Universal Robots PolyScope program: p1kine.urp

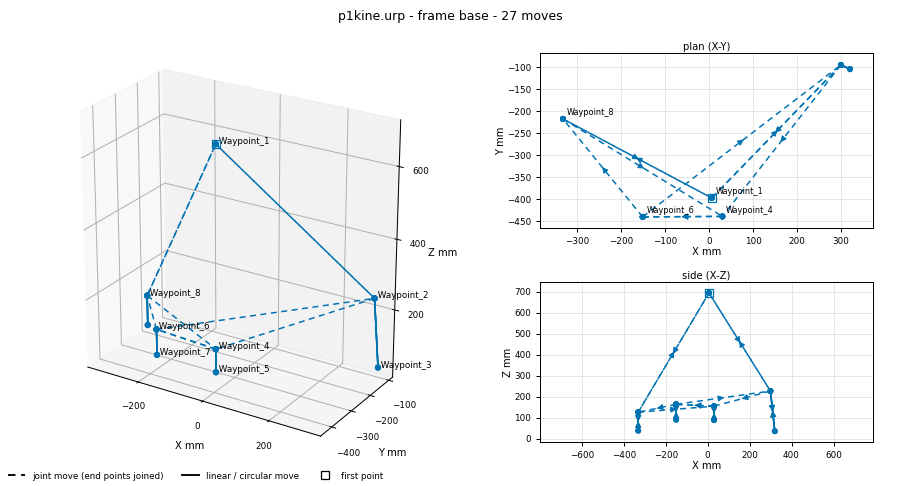
[picture p0: tool path of p1kine.urp in frame base, 27 of 27 moves have a stored position in this frame; points joined in program order, loops and branches not executed]
Program p1kine (installation=default directory=/programs createdIn=5.14.5 lastSavedIn=5.14.5 robotSerialNumber=20195300809)
Calibrated DH parameters: a=[-0.000085, -0.20076, -0.212369, 0.000121, -0.000118, 0]; d=[0.15185, -26.306375, 24.753047, 1.684739, 0.085386, 0.092088]; alpha=[1.572149, -0.00522, -0.011864, 1.571339, -1.571085, 0]; deltaTheta=[0, 0.599885, -0.513355, -0.086555, 0.000006, 0]
InitVariablesNode
Robot Program (runOnlyOnce=false)
  'Make sure gripper open'
  URCap Gripper Activate (Robotiq_Grippers, Robotiq Inc.) dataModel(ResetAndActivateKey=false)
  URCap Gripper (Robotiq_Grippers, Robotiq Inc.) dataModel(position=0.0, force=0.0, speed=100.0, positionInDouble=0.0, forceInDouble=0.0, speedInDouble=100.0, slaveIds=[9], blocking=true)
  Wait Sleep waitTime=1
  MoveJ speed 60 deg/s, acceleration 80 deg/s^2 (useActiveTCP=true) feature=Base
    Waypoint Waypoint_1: TCP in base x=6.371 y=-396.697 z=694.74 mm, rx=-0.018 ry=2.2102 rz=-2.2165 rad; joints [0.003, -90.002, 0, -90.003, 0.001, 0.002] deg; TCP offset x=0 y=0 z=174 mm, rx=0 ry=0 rz=0 rad
  Wait Sleep waitTime=0.5
  MoveJ speed 60 deg/s, acceleration 80 deg/s^2 (useActiveTCP=true) feature=Base
    Waypoint Waypoint_2: TCP in base x=299.3 y=-94.865 z=226.793 mm, rx=-3.1332 ry=0.0855 rz=-0.0071 rad; joints [6.366, -92.288, -60.191, -117.184, 89.878, -79.859] deg
    MoveL speed 250 mm/s, acceleration 1200 mm/s^2 (useActiveTCP=true) feature=Base
      Waypoint Waypoint_3: TCP in base x=320.061 y=-104.261 z=35.408 mm, rx=3.0968 ry=0.0304 rz=0.0101 rad; joints [6.956, -96.302, -109.066, -64.528, 86.845, -84.116] deg
      URCap Gripper (Robotiq_Grippers, Robotiq Inc.) dataModel(position=100.0, force=0.0, speed=100.0, positionInDouble=100.0, forceInDouble=0.0, speedInDouble=100.0, slaveIds=[9], blocking=true)
    MoveL speed 250 mm/s, acceleration 1200 mm/s^2 (useActiveTCP=true) feature=Base
      Waypoint Waypoint_2: TCP in base x=299.3 y=-94.865 z=226.793 mm, rx=-3.1332 ry=0.0855 rz=-0.0071 rad; joints [6.366, -92.288, -60.191, -117.184, 89.878, -79.859] deg
    MoveJ speed 60 deg/s, acceleration 80 deg/s^2 (useActiveTCP=true) feature=Base
      Waypoint Waypoint_4: TCP in base x=30.368 y=-438.454 z=154.559 mm, rx=2.1917 ry=-2.2123 rz=0.0571 rad; joints [-68.558, -117.991, -48.054, -101.406, 88.704, -67.517] deg
      MoveL speed 250 mm/s, acceleration 1200 mm/s^2 (useActiveTCP=true) feature=Base
        Waypoint Waypoint_5: TCP in base x=30.354 y=-438.451 z=88.458 mm, rx=2.2337 ry=-2.2072 rz=0.0186 rad; joints [-69.045, -119.099, -63.398, -86.835, 89.483, -69.377] deg
        URCap Gripper (Robotiq_Grippers, Robotiq Inc.) dataModel(position=0.0, force=0.0, speed=100.0, positionInDouble=0.0, forceInDouble=0.0, speedInDouble=100.0, slaveIds=[9], blocking=true)
      MoveL speed 250 mm/s, acceleration 1200 mm/s^2 (useActiveTCP=true) feature=Base
        Waypoint Waypoint_4: TCP in base x=30.368 y=-438.454 z=154.559 mm, rx=2.1917 ry=-2.2123 rz=0.0571 rad; joints [-68.558, -117.991, -48.054, -101.406, 88.704, -67.517] deg
        Wait Sleep waitTime=2
        Set DigitalOutput pin=digital_out[0]; digitalValue=1
        Wait DigitalInput pin=digital_in[0]; digitalValue=0
        Set Undefined
        Set DigitalOutput pin=digital_out[0]; digitalValue=0
    MoveJ speed 60 deg/s, acceleration 80 deg/s^2 (useActiveTCP=true) feature=Base
      Waypoint Waypoint_6: TCP in base x=-150.595 y=-439.593 z=163.821 mm, rx=2.2337 ry=-2.2073 rz=0.0186 rad; joints [-93.029, -136.008, -12.994, -120.473, 89.767, -92.991] deg
    MoveL speed 250 mm/s, acceleration 1200 mm/s^2 (useActiveTCP=true) feature=Base
      Waypoint Waypoint_7: TCP in base x=-150.303 y=-439.589 z=90.363 mm, rx=2.2338 ry=-2.2072 rz=0.0186 rad; joints [-92.983, -126.706, -50.488, -92.283, 89.694, -93.25] deg
    URCap Gripper (Robotiq_Grippers, Robotiq Inc.) dataModel(position=100.0, force=0.0, speed=100.0, positionInDouble=100.0, forceInDouble=0.0, speedInDouble=100.0, slaveIds=[9], blocking=true)
    MoveL speed 250 mm/s, acceleration 1200 mm/s^2 (useActiveTCP=true) feature=Base
      Waypoint Waypoint_6: TCP in base x=-150.595 y=-439.593 z=163.821 mm, rx=2.2337 ry=-2.2073 rz=0.0186 rad; joints [-93.029, -136.008, -12.994, -120.473, 89.767, -92.991] deg
    MoveJ speed 60 deg/s, acceleration 80 deg/s^2 (useActiveTCP=true) feature=Base
      Waypoint Waypoint_8: TCP in base x=-331.355 y=-217.265 z=126.037 mm, rx=-1.3074 ry=2.8357 rz=-0.0113 rad; joints [-128.298, -109.343, -67.085, -94.331, 90.198, -87.379] deg
    MoveL speed 250 mm/s, acceleration 1200 mm/s^2 (useActiveTCP=true) feature=Base
      Waypoint Waypoint_9: TCP in base x=-331.352 y=-217.234 z=37.633 mm, rx=-1.3074 ry=2.8356 rz=-0.0113 rad; joints [-128.237, -112.383, -86.934, -71.449, 90.193, -87.583] deg
    URCap Gripper (Robotiq_Grippers, Robotiq Inc.) dataModel(position=0.0, force=0.0, speed=0.0, positionInDouble=0.0, forceInDouble=0.0, speedInDouble=0.0, slaveIds=[9], blocking=true)
    MoveL speed 250 mm/s, acceleration 1200 mm/s^2 (useActiveTCP=true) feature=Base
      Waypoint Waypoint_8: TCP in base x=-331.355 y=-217.265 z=126.037 mm, rx=-1.3074 ry=2.8357 rz=-0.0113 rad; joints [-128.298, -109.343, -67.085, -94.331, 90.198, -87.379] deg
  MoveJ speed 60 deg/s, acceleration 80 deg/s^2 (useActiveTCP=true) feature=Base
    Waypoint Waypoint_10: TCP in base x=6.326 y=-396.697 z=694.74 mm, rx=-0.0179 ry=2.2102 rz=-2.2166 rad; joints [-0.001, -90, 0, -90, 0, -0.004] deg
    Wait Sleep waitTime=1
    Waypoint Waypoint_8: TCP in base x=-331.355 y=-217.265 z=126.037 mm, rx=-1.3074 ry=2.8357 rz=-0.0113 rad; joints [-128.298, -109.343, -67.085, -94.331, 90.198, -87.379] deg
  MoveL speed 250 mm/s, acceleration 1200 mm/s^2 (useActiveTCP=true) feature=Base
    Waypoint Waypoint_9: TCP in base x=-331.352 y=-217.234 z=37.633 mm, rx=-1.3074 ry=2.8356 rz=-0.0113 rad; joints [-128.237, -112.383, -86.934, -71.449, 90.193, -87.583] deg
    URCap Gripper (Robotiq_Grippers, Robotiq Inc.) dataModel(position=100.0, force=0.0, speed=100.0, positionInDouble=100.0, forceInDouble=0.0, speedInDouble=100.0, slaveIds=[9], blocking=true)
    Wait Sleep waitTime=1
    Waypoint Waypoint_8: TCP in base x=-331.355 y=-217.265 z=126.037 mm, rx=-1.3074 ry=2.8357 rz=-0.0113 rad; joints [-128.298, -109.343, -67.085, -94.331, 90.198, -87.379] deg
  MoveJ speed 60 deg/s, acceleration 80 deg/s^2 (useActiveTCP=true) feature=Base
    Waypoint Waypoint_4: TCP in base x=30.368 y=-438.454 z=154.559 mm, rx=2.1917 ry=-2.2123 rz=0.0571 rad; joints [-68.558, -117.991, -48.054, -101.406, 88.704, -67.517] deg
  MoveL speed 250 mm/s, acceleration 1200 mm/s^2 (useActiveTCP=true) feature=Base
    Waypoint Waypoint_5: TCP in base x=30.354 y=-438.451 z=88.458 mm, rx=2.2337 ry=-2.2072 rz=0.0186 rad; joints [-69.045, -119.099, -63.398, -86.835, 89.483, -69.377] deg
    URCap Gripper (Robotiq_Grippers, Robotiq Inc.) dataModel(position=0.0, force=0.0, speed=100.0, positionInDouble=0.0, forceInDouble=0.0, speedInDouble=100.0, slaveIds=[9], blocking=true)
  MoveL speed 250 mm/s, acceleration 1200 mm/s^2 (useActiveTCP=true) feature=Base
    Waypoint Waypoint_4: TCP in base x=30.368 y=-438.454 z=154.559 mm, rx=2.1917 ry=-2.2123 rz=0.0571 rad; joints [-68.558, -117.991, -48.054, -101.406, 88.704, -67.517] deg
    Wait Sleep waitTime=2
    Set DigitalOutput pin=digital_out[0]; digitalValue=1
    Wait DigitalInput pin=digital_in[0]; digitalValue=0
    Set DigitalOutput pin=digital_out[0]; digitalValue=0
  MoveJ speed 60 deg/s, acceleration 80 deg/s^2 (useActiveTCP=true) feature=Base
    Waypoint Waypoint_6: TCP in base x=-150.595 y=-439.593 z=163.821 mm, rx=2.2337 ry=-2.2073 rz=0.0186 rad; joints [-93.029, -136.008, -12.994, -120.473, 89.767, -92.991] deg
  MoveL speed 250 mm/s, acceleration 1200 mm/s^2 (useActiveTCP=true) feature=Base
    Waypoint Waypoint_7: TCP in base x=-150.303 y=-439.589 z=90.363 mm, rx=2.2338 ry=-2.2072 rz=0.0186 rad; joints [-92.983, -126.706, -50.488, -92.283, 89.694, -93.25] deg
  URCap Gripper (Robotiq_Grippers, Robotiq Inc.) dataModel(position=100.0, force=0.0, speed=100.0, positionInDouble=100.0, forceInDouble=0.0, speedInDouble=100.0, slaveIds=[9], blocking=true)
  MoveL speed 250 mm/s, acceleration 1200 mm/s^2 (useActiveTCP=true) feature=Base
    Waypoint Waypoint_6: TCP in base x=-150.595 y=-439.593 z=163.821 mm, rx=2.2337 ry=-2.2073 rz=0.0186 rad; joints [-93.029, -136.008, -12.994, -120.473, 89.767, -92.991] deg
  MoveJ speed 60 deg/s, acceleration 80 deg/s^2 (useActiveTCP=true) feature=Base
    Waypoint Waypoint_2: TCP in base x=299.3 y=-94.865 z=226.793 mm, rx=-3.1332 ry=0.0855 rz=-0.0071 rad; joints [6.366, -92.288, -60.191, -117.184, 89.878, -79.859] deg
  MoveL speed 250 mm/s, acceleration 1200 mm/s^2 (useActiveTCP=true) feature=Base
    Waypoint Waypoint_3: TCP in base x=320.061 y=-104.261 z=35.408 mm, rx=3.0968 ry=0.0304 rz=0.0101 rad; joints [6.956, -96.302, -109.066, -64.528, 86.845, -84.116] deg
    URCap Gripper (Robotiq_Grippers, Robotiq Inc.) dataModel(position=0.0, force=0.0, speed=100.0, positionInDouble=0.0, forceInDouble=0.0, speedInDouble=100.0, slaveIds=[9], blocking=true)
    Wait Sleep waitTime=1
    Waypoint Waypoint_2: TCP in base x=299.3 y=-94.865 z=226.793 mm, rx=-3.1332 ry=0.0855 rz=-0.0071 rad; joints [6.366, -92.288, -60.191, -117.184, 89.878, -79.859] deg
  MoveJ speed 60 deg/s, acceleration 80 deg/s^2 (useActiveTCP=true) feature=Base
    Waypoint Waypoint_11: TCP in base x=6.335 y=-396.697 z=694.74 mm, rx=-0.018 ry=2.2102 rz=-2.2166 rad; joints [0, -90.001, 0.002, -90.004, -0.001, -0.002] deg
